(* 	Disclaimer
	All sample code provided by Beckhoff Automation LLC are for illustrative purposes only and are provided “as is” and without any warranties, express or implied.
	Actual implementations in applications will vary significantly.
	Beckhoff Automation LLC shall have no liability for, and does not waive any rights in relation to, any code samples that it provides or the use of such code samples for any purpose.
*)
FUNCTION_BLOCK FB_Debounce
VAR_INPUT
	In: BOOL;
	TimeOn: TIME := T#2S;
	TimeOff: TIME := T#2S;
END_VAR
VAR_OUTPUT
	Out: BOOL;
END_VAR
VAR
	tonDelayOn: TON;
	tonDelayOff: TON;
END_VAR

// Set-Reset delay Timers
IF In THEN
	tonDelayOn.PT := TimeOn;
	tonDelayOn.IN := TRUE;
	tonDelayOff.IN := FALSE;
ELSE
	tonDelayOff.PT := TimeOff;
	tonDelayOff.IN := TRUE;
	tonDelayOn.IN := FALSE;
END_IF

// Set delayed Output
IF tonDelayOn.Q THEN
	Out := TRUE;
END_IF

// Reset delayed Output
IF tonDelayOff.Q THEN
	Out := FALSE;
END_IF

// Call function blocks
tonDelayOn();
tonDelayOff();

END_FUNCTION_BLOCK

(* stored: Version 1.1.0.1, ProductVersion 3.1.4024.12
   POU FB_Debounce: Id {6e938fe1-dd2a-4782-a13d-85026131fc45}, SpecialFunc None *)
